# EPICS substitutions: iocBoot/ioc6idACS1/substitutions/canberra_13.substitutions
file "$(MCA)/mcaApp/Db/simple_mca.db"
{
pattern
{P           M       DTYP           INP         PREC  CHANS}
{6idACS1:med:   mca1  "asynMCA"   "@asyn(AIM2/1 0)"    3  2048}
{6idACS1:med:   mca2  "asynMCA"   "@asyn(AIM2/1 1)"    3  2048}
{6idACS1:med:   mca3  "asynMCA"   "@asyn(AIM2/1 2)"    3  2048}
{6idACS1:med:   mca4  "asynMCA"   "@asyn(AIM2/2 0)"    3  2048}
{6idACS1:med:   mca5  "asynMCA"   "@asyn(AIM2/2 1)"    3  2048}
{6idACS1:med:   mca6  "asynMCA"   "@asyn(AIM2/2 2)"    3  2048}
{6idACS1:med:   mca7  "asynMCA"   "@asyn(AIM3/1 0)"    3  2048}
{6idACS1:med:   mca8  "asynMCA"   "@asyn(AIM3/1 1)"    3  2048}
{6idACS1:med:   mca9  "asynMCA"   "@asyn(AIM3/1 2)"    3  2048}
{6idACS1:med:   mca10 "asynMCA"   "@asyn(AIM3/2 0)"    3  2048}
{6idACS1:med:   mca11 "asynMCA"   "@asyn(AIM3/3 1)"    3  2048}
{6idACS1:med:   mca12 "asynMCA"   "@asyn(AIM3/4 2)"    3  2048}
{6idACS1:med:   mca13 "asynMCA"   "@asyn(AIM3/2 3)"    3  2048}
{6idACS1:med:   mca0  "Soft Channel"   ""     3  2048}
}

file "$(MCA)/mcaApp/Db/icb_amp.db"
{
pattern
{P			AMP		PORT}
{6idACS1:med:	amp1	"icbAmp1"}
{6idACS1:med:	amp2	"icbAmp2"}
{6idACS1:med:	amp3	"icbAmp3"}
{6idACS1:med:	amp4	"icbAmp4"}
{6idACS1:med:	amp5	"icbAmp5"}
{6idACS1:med:	amp6	"icbAmp6"}
{6idACS1:med:	amp7	"icbAmp7"}
{6idACS1:med:	amp8	"icbAmp8"}
{6idACS1:med:	amp9	"icbAmp9"}
{6idACS1:med:	amp10	"icbAmp10"}
{6idACS1:med:	amp11	"icbAmp11"}
{6idACS1:med:	amp12	"icbAmp12"}
{6idACS1:med:	amp13	"icbAmp13"}
}

file "$(MCA)/mcaApp/Db/icb_adc.db"
{
pattern
{P			ADC		PORT}
{6idACS1:med:	adc1	"icbAdc1"}
{6idACS1:med:	adc2	"icbAdc2"}
{6idACS1:med:	adc3	"icbAdc3"}
{6idACS1:med:	adc4	"icbAdc4"}
}

file "$(MCA)/mcaApp/Db/icb_hvps.db"
{
pattern
{P			HVPS	LIMIT	PORT}
{6idACS1:med:	hvps1	1000	"icbHvps1"}
}
